FUNCTION_BLOCK TXml EXTENDS TExecution
VAR_INPUT
	FilePath : T_MaxString;
	XPath 	 : T_MaxString;
	AddHeaderNodeXml : PVOID;
	SizeOfHeaderNodeXml : UDINT;
END_VAR
VAR_OUTPUT	
END_VAR
VAR
	{attribute 'hide'}		  
	{attribute 'OPC.UA.DA' := '0'}
	_xmlSrvRead : FB_XmlSrvRead;			
	{attribute 'OPC.UA.DA' := '0'}
	_deserialisationOperation : TExecution;	
	{attribute 'OPC.UA.DA' := '0'}
	item : INT;
	{attribute 'OPC.UA.DA' := '0'}
	_logger : Logger;
	{attribute 'OPC.UA.DA' := '0'}
	_message : StringBuilder;
END_VAR

Deserialize(_deserialisationOperation.Starting);

IF _xmlSrvRead.bBusy THEN
    _deserialisationOperation.SetBusy();
END_IF

IF _xmlSrvRead.bError THEN
	_deserialisationOperation.SetError(ErrorId := _xmlSrvRead.nErrId);
		
	_logger.Error(_message.Reset().Append('Xml deserialization - ErrorId : ').
			 			   		   Append(UDINT_TO_STRING(_xmlSrvRead.nErrId)).ToString());
END_IF 

IF _deserialisationOperation.Busy THEN
    IF NOT _xmlSrvRead.bBusy THEN        
        IF THIS^.Aborted THEN
            _deserialisationOperation.SetAborted();
			_logger.Information(_message.Reset().Append('Xml deserialization aborted').ToString());
        ELSE
            _deserialisationOperation.SetDone(); 
			_logger.Debug(_message.Reset().Append('Xml deserialization done').ToString());
        END_IF
    END_IF
END_IF

PROPERTY DeserialisationOperation : IExecution
GET
DeserialisationOperation := _deserialisationOperation;
END_GET
END_PROPERTY

METHOD Deserialize
VAR_INPUT
	Execute : BOOL;
END_VAR
CASE item OF
0:
	IF Execute THEN
		THIS^.State := TExecutionState.Busy;
		_logger.Debug(_message.Reset().Append('Xml deserialization busy').ToString());
		item := item + 1;
	END_IF
1:	
	_xmlSrvRead(
	  pSymAddr	:= AddHeaderNodeXml,
	  cbSymSize	:= SizeOfHeaderNodeXml, 
	  sFilePath	:= FilePath,
	  sXPath	:= XPath,
	  bExecute	:= TRUE
	);	
	item := item + 1;	
		
2:  
	_xmlSrvRead(bExecute:= FALSE);
	IF NOT _xmlSrvRead.bBusy AND NOT _xmlSrvRead.bError THEN		
		THIS^.State := TExecutionState.Ready;
		item := 0;
	END_IF	
END_CASE
END_METHOD

END_FUNCTION_BLOCK

(* stored: Version 1.1.0.1, ProductVersion 3.1.4024.3
   POU TXml: Id {8ed1d49a-ee13-479c-b8cf-ad238d58e526}, SpecialFunc None
   Property DeserialisationOperation: Id {b89debbd-8683-487c-a555-8b5b730c00d8}
   Get Get: Id {3f64bf07-c8f2-4dcf-a39d-df45e934e828}
   Method Deserialize: Id {534256e8-5203-4668-ad42-05cb4e102d28} *)
